TYPE ST_ProductData :
STRUCT
	bPass				:BOOL;
	bFail				:BOOL;
END_STRUCT
END_TYPE

(* stored: Version 1.1.0.1, ProductVersion 3.1.4024.10
   DUT ST_ProductData: Id {cf6a5e28-71b9-4746-8cf0-ea891c5c3d84} *)
